{attribute 'linkalways'} 
{attribute 'no_explicit_call' := 'This FB is a CLASS and must be accessed using methods or properties'}
{attribute 'enable_dynamic_creation'}
FUNCTION_BLOCK IncorrectTypeDeserializationError EXTENDS Error
VAR
	dataType : T_MAXSTRING;
END_VAR

PROPERTY PUBLIC ErrorType : T_MAXSTRING
GET
ErrorType := 'INCORRECT_DATATYPE_DESERIALIZATION_ERROR';
END_GET
END_PROPERTY

METHOD FB_init : BOOL
VAR_INPUT
	bInitRetains : BOOL; // if TRUE, the retain variables are initialized (warm start / cold start)
	bInCopyCode : BOOL;  // if TRUE, the instance afterwards gets moved into the copy code (online change)
	DataType : T_MAXSTRING;
END_VAR
THIS^.dataType := DataType;
END_METHOD

PROPERTY PUBLIC Message : T_MAXSTRING
GET
Message := CONCAT('Deserialization Failed, Incorrect Datatype : ', dataType);
END_GET
END_PROPERTY

END_FUNCTION_BLOCK

(* stored: Version 1.1.0.1, ProductVersion 3.1.4024.12
   POU IncorrectTypeDeserializationError: Id {dc907ea0-6a28-0b98-0c9e-d21873a1d86a}, SpecialFunc None
   Folder Constructor: Id {ace4d44a-dce7-08a6-0c50-b921072d34f6}
   Property ErrorType: Id {9a3b4d8d-035c-067b-3f53-a8c5d6098c08}
   Get Get: Id {f92dac36-1548-04ed-3aa7-626c8d81b5ce}
   Method FB_init: Id {c64dc449-230e-002a-016f-edde0580e173}
   Property Message: Id {53a7e599-0c76-0043-186f-2abf7843b052}
   Get Get: Id {cb60782a-5925-0d1a-1691-24587a8558f6} *)
